FUNCTION FSum : dint
VAR_IN_OUT
    aData     : ARRAY [*] OF INT;
END_VAR
VAR
    i, nSum   : DINT;
END_VAR

nSum := 0;
 
FOR i := LOWER_BOUND(aData,1) TO UPPER_BOUND(aData,1) DO
    nSum := nSum + aData[i];
END_FOR;

FSum := nSum;

END_FUNCTION

(* stored: Version 1.1.0.1, ProductVersion 3.1.4024.12
   POU FSum: Id {6bee12a3-ac00-4502-acf5-cdc9cd51b9e2}, SpecialFunc None *)
